FUNCTION_BLOCK TL_CentrContr (* Composite Function Block Type *)
  (* Standard: 61499-2 *)
  (* Version 0.2, 2003-12-05, JHC, Rockwell Automation, Renamed from NEWCOMPFB. *)
  (* Version 0.1, 2002-01-08, JHC, Rockwell Automation, Added DLY FB as example. *)
  (* Version 0.0, 2000-05-27, JHC, Rockwell Automation *)
  PACKAGE fb.rt.template;
  IMPORT fb.datatype.*;
  IMPORT fb.rt.*;
  IMPORT fb.rt.myfb.TLCtrl;
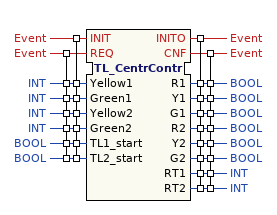
  EVENT_INPUT
    INIT WITH Yellow1, Green1, Yellow2, Green2, TL1_start, TL2_start; (* Initialization Request *)
    REQ WITH Yellow1, Green1, Yellow2, Green2, TL1_start, TL2_start; (* Normal Execution Request *)
  END_EVENT
  EVENT_OUTPUT
    INITO WITH R1, Y1, G1, R2, G2, Y2, RT1, RT2; (* Initialization Confirm *)
    CNF WITH R1, Y1, G1, R2, Y2, G2, RT1, RT2; (* Execution Confirmation *)
  END_EVENT
  VAR_INPUT
    Yellow1 : INT;
    Green1 : INT;
    Yellow2 : INT;
    Green2 : INT;
    TL1_start : BOOL;
    TL2_start : BOOL;
  END_VAR
  VAR_OUTPUT
    R1 : BOOL;
    Y1 : BOOL;
    G1 : BOOL;
    R2 : BOOL;
    Y2 : BOOL;
    G2 : BOOL;
    RT1 : INT;
    RT2 : INT;
  END_VAR
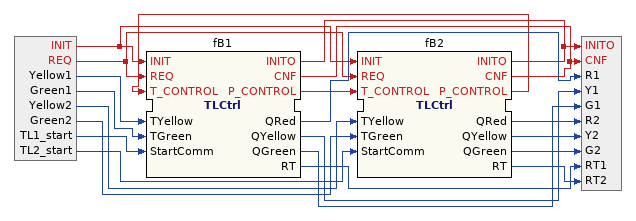
  FBS
    fB1 : TLCtrl;
    fB2 : TLCtrl;
  END_FBS
  EVENT_CONNECTIONS
    fB1.P_CONTROL TO fB2.T_CONTROL;
    fB2.P_CONTROL TO fB1.T_CONTROL;
    INIT TO fB1.INIT;
    REQ TO fB1.REQ;
    fB2.INITO TO INITO;
    fB2.CNF TO CNF;
    REQ TO fB2.REQ;
    fB1.CNF TO CNF;
    INIT TO fB2.INIT;
    fB1.INITO TO INITO;
  END_CONNECTIONS
  DATA_CONNECTIONS
    Yellow1 TO fB1.TYellow;
    Green1 TO fB1.TGreen;
    TL1_start TO fB1.StartComm;
    Yellow2 TO fB2.TYellow;
    Green2 TO fB2.TGreen;
    TL2_start TO fB2.StartComm;
    fB1.QRed TO R1;
    fB1.QYellow TO Y1;
    fB1.QGreen TO G1;
    fB2.QRed TO R2;
    fB2.QYellow TO Y2;
    fB2.QGreen TO G2;
    fB1.RT TO RT1;
    fB2.RT TO RT2;
  END_CONNECTIONS
END_FUNCTION_BLOCK
